TYPE ST_DALI103Parameters :
STRUCT
	nOperatingMode			:	BYTE;
	sInstanceType0			:	STRING;
	sInstanceType1			:	STRING;
	sInstanceType2			:	STRING;
	sInstanceType3			:	STRING;
	sInstanceType4			:	STRING;
END_STRUCT
END_TYPE

(* stored: Version 1.1.0.1, ProductVersion 3.1.4024.12
   DUT ST_DALI103Parameters: Id {63db6246-0618-4ff9-be19-67e8ef4dbe28} *)
